// TIA Portal V19 export
TYPE "LEXCHANGETRAY_typePlasticEm5_interface"
// stored: Access Published
   STRUCT
      deliver : "LEXCHANGETRAY_typePlasticEm5_deliver_interface";
      recieve : "LEXCHANGETRAY_typePlasticEm5_recieve_interface";
   END_STRUCT;
END_TYPE
